FUNCTION_BLOCK FB_ParamSaveRestoreNC_TestDouble IMPLEMENTS I_ParamSaveRestore
VAR_INPUT
END_VAR
VAR_OUTPUT
END_VAR
VAR
END_VAR

{warning 'Add property implementation'}
PROPERTY Aborted : BOOL
GET
END_GET
END_PROPERTY

{warning 'Add property implementation'}
PROPERTY Active : BOOL
GET
END_GET
END_PROPERTY

{warning 'Add property implementation'}
PROPERTY Busy : BOOL
GET
END_GET
END_PROPERTY

{warning 'Add property implementation'}
PROPERTY Done : BOOL
GET
END_GET
END_PROPERTY

{warning 'Add property implementation'}
PROPERTY Error : BOOL
GET
END_GET
END_PROPERTY

{warning 'Add property implementation'}
PROPERTY ErrorID : UDINT
GET
END_GET
END_PROPERTY

{warning 'Add property implementation'}
PROPERTY Message : T_MAXSTRING
GET
END_GET
END_PROPERTY

{warning 'Add method implementation '}
METHOD RestoreAxisParams
END_METHOD

{warning 'Add method implementation '}
METHOD SaveAxisParams
VAR_INPUT
    Enable	: BOOL;
END_VAR
END_METHOD

{warning 'Add property implementation'}
PROPERTY SavedPosition : LREAL
GET
END_GET
END_PROPERTY

END_FUNCTION_BLOCK

(* stored: Version 1.1.0.1
   POU FB_ParamSaveRestoreNC_TestDouble: Id {634c36c5-150a-4764-a0a6-c7ecdf090bad}, SpecialFunc None
   Property Aborted: Id {dfc73d04-88ad-4e3f-a76e-a62be28f51db}
   Get Get: Id {312de29d-84e3-4d8a-98a8-ac5bbc7581e2}
   Property Active: Id {50d7dceb-cfc3-4a07-91b2-df0929c39447}
   Get Get: Id {afdf8856-06a6-40a4-a2bc-2d946980885f}
   Property Busy: Id {0b1afbf6-91b2-4368-96d9-d83740a58dcc}
   Get Get: Id {a25ce8e7-6949-465e-bca1-574968b6c23e}
   Property Done: Id {970ebffa-50ba-4340-b875-23a06b5b2f5e}
   Get Get: Id {ee36213a-2801-45a7-afc0-333d7ef8e430}
   Property Error: Id {c0783019-d820-4692-872e-61757b758b78}
   Get Get: Id {936b8fed-7a2f-414d-a7f5-2bfa436b6dfb}
   Property ErrorID: Id {38508d52-346a-4ddd-af00-ed74ba87a1c0}
   Get Get: Id {d8077fba-7f1f-48ba-a78b-c1450d72e9d0}
   Property Message: Id {03cb698e-097b-41de-8e43-d25d618343c1}
   Get Get: Id {c4bf9478-03b2-4cce-9ac5-9a1b7b5bdfbc}
   Method RestoreAxisParams: Id {437fdd5e-5302-485c-a780-b9bb9a2bb27d}
   Method SaveAxisParams: Id {279440a3-1ce4-42ac-9234-61b3894a0684}
   Property SavedPosition: Id {a013de21-964c-4969-845c-335038b9278b}
   Get Get: Id {a55681bf-1d9e-4fad-af00-a74243a38447} *)
